FUNCTION_BLOCK fb_Worker
VAR
  _nProcess         : UINT;

  _ItfProcess       : REFERENCE TO ARRAY[1..MAX_PROCESS] OF I_ExternControl_Process;

  _tonProcess       : Tc2_Standard.TON;
  _tProcess         : TIME;

  _nMoverPerMinute  : UINT;

  _wTargetMask      : DWORD;
  _nQueue           : ARRAY[1..MAX_PROCESS] OF UINT;

END_VAR

METHOD AUTO : E_PROGRESS
VAR_INPUT
  Active            : BOOL;
END_VAR
VAR_INST
  _bSparse            : Bool;
  _ncount             : uint;
  _eState,
  _eResult            : E_PROGRESS;

  _ndx                : UINT;

  _eProcessState      : E_STATION_STATE;
  _eProcessCmd        : E_STATION_CTRL;

  _nkx                : UINT;

  _nInputLastTarget   : UINT;

{attribute 'displaymode':='bin'}
  _wBufferSentMask    : dword;
{attribute 'displaymode':='bin'}
  _wProcessInputMask  : dWORD; // placement information for movers in stations from preceeding machine
END_VAR
IF NOT Check() THEN AUTO := E_PROGRESS.PROGRESS_ERROR; RETURN; END_IF

//-----------------------------------------------------------------------------
IF NOT Active 
THEN 
	_eState                                     := E_PROGRESS.PROGRESS_INIT;

  _nCount                                     := 0;
  memset(ADR(_nQueue), 0, SIZEOF(_nQueue));
  memset(ADR(_wProcessInputMask), 0, SIZEOF(_wProcessInputMask));
  memset(ADR(_wBufferSentMask), 0, SIZEOF(_wBufferSentMask));
ELSE
  _eProcessState                              := _ItfProcess[_nProcess].ProcessState;

  FOR _ndx := 1 TO MAX_PROCESS
  DO
    _nQueue[_ndx]                             := _ItfProcess[_ndx].MoverCountInQueue;
  END_FOR
END_IF 
//-----------------------------------------------------------------------------
//-----------------------------------------------------------------------------
//-----------------------------------------------------------------------------
CASE _eState
OF
  E_PROGRESS.PROGRESS_INIT:
    IF Active
    THEN
      _nCount := _ncount + 1;
      _wProcessInputMask                      := 0;
      _wBufferSentMask                        := 0;
      _eState                                 := E_PROGRESS.PROGRESS_BUSY;
    END_IF
END_CASE
//-----------------------------------------------------------------------------
//-----------------------------------------------------------------------------
CASE _eState
OF
  E_PROGRESS.PROGRESS_BUSY:

    CASE _nProcess
    OF
      DISTRIBUTOR_2,
      DISTRIBUTOR_1:
        _eState                               := E_PROGRESS.PROGRESS_PREPARE;

      OUTPUT_R2:
        _eState                               := E_PROGRESS.PROGRESS_PREPARE;

      OUTPUT_R1:
        _eState                               := E_PROGRESS.PROGRESS_PREPARE;

      BUFFER_3:
        IF (_nQueue[BUFFER_3] > QUEUE_COUNT)
        THEN
          _eState                             := E_PROGRESS.PROGRESS_PREPARE;
        END_IF

      OUTPUT_1:
        _eState                               := E_PROGRESS.PROGRESS_PREPARE;

      INPUT:
        _eState                               := E_PROGRESS.PROGRESS_PREPARE;

      BUFFER_1:
        _eState                               := E_PROGRESS.PROGRESS_PREPARE;
        IF NOT _bSparse
        THEN
          FOR _nkx := 1 TO _ItfProcess[INPUT].StationCount
          DO
              _wProcessInputMask              := Tc2_System.SETBIT32(_wProcessInputMask, TO_SINT(_nkx-1));
          END_FOR
        ELSE
          FOR _nkx := 1 TO _ItfProcess[INPUT].StationCount
          DO
            IF (_nkx <> 7)
            THEN
              _wProcessInputMask              := _ItfProcess[BUFFER_1].SetBitDWord(_wProcessInputMask, _nkx-1);
            END_IF
          END_FOR

        END_IF


      BUFFER_4:
        IF (_nQueue[BUFFER_1] < 8)
        THEN
          _eState                             := E_PROGRESS.PROGRESS_PREPARE;
        END_IF
    END_CASE
END_CASE
//-----------------------------------------------------------------------------
//-----------------------------------------------------------------------------
CASE _eState
OF
  E_PROGRESS.PROGRESS_PREPARE:
    CASE _nProcess
    OF
      BUFFER_1:
        _bSparse                              := FALSE;
        IF (_nQueue[INPUT] = 0)
        THEN
          _nInputLastTarget                   := 0;
          _ItfProcess[BUFFER_1].TargetMask    := _wProcessInputMask;
          _eState                             := E_PROGRESS.PROGRESS_WORKING;
        END_IF
    ELSE
      _eState                                 := E_PROGRESS.PROGRESS_WORKING;
    END_CASE

END_CASE
//-----------------------------------------------------------------------------
//-----------------------------------------------------------------------------
CASE _eState
OF
  E_PROGRESS.PROGRESS_WORKING:

  CASE _eProcessState
  OF
    E_STATION_STATE.STATION_INIT:
      CASE _nProcess
      OF
        BUFFER_3:
          IF (_nQueue[OUTPUT_R1] = QUEUE_COUNT)
          THEN
            _eState                           := E_PROGRESS.PROGRESS_INIT;
          ELSE
            _eProcessCmd                      := E_STATION_CTRL.STATION_DISABLE;
          END_IF
      ELSE
        _eProcessCmd                          := E_STATION_CTRL.STATION_DISABLE;
      END_CASE

    E_STATION_STATE.STATION_DISABLE:
      _eProcessCmd                            := E_STATION_CTRL.STATION_ENABLE;

    E_STATION_STATE.STATION_MOVER_ENTER:
      CASE _ItfProcess[_nProcess].ProcessType
      OF
        E_PROCESS_TYPE.DISTRIBUTOR:
          IF (GVL_XTS.StationState[_ItfProcess[_nProcess].StationFirst].rMoverModPos > GVL_XTS.StationParameter[_ItfProcess[_nProcess].StationFirst].rPosWait-5.0)
          THEN
            _eState                           := E_PROGRESS.PROGRESS_OCCUPIED;
            _eProcessCmd                      := E_STATION_CTRL.STATION_MOVER_SEND;
          END_IF
      ELSE
          _eProcessCmd                        := E_STATION_CTRL.STATION_MOVER_ENTER;
      END_CASE

    E_STATION_STATE.STATION_PROCESS_START:
      _tonProcess(IN := FALSE, PT := _tProcess);
      CASE _nProcess
      OF
        INPUT:
          IF (_nQueue[INPUT] = QUEUE_COUNT)
          THEN
            _eProcessCmd                      := E_STATION_CTRL.STATION_PROCESS_START;
          END_IF

        OUTPUT_R1,
        OUTPUT_R2:
          IF (_ItfProcess[OUTPUT_R1].ProcessState = _ItfProcess[OUTPUT_R2].ProcessState)
          THEN
            _eProcessCmd                      := E_STATION_CTRL.STATION_PROCESS_START;
          END_IF
      ELSE
        _eProcessCmd                          := E_STATION_CTRL.STATION_PROCESS_START;
      END_CASE


    E_STATION_STATE.STATION_PROCESS_DONE:
      _tonProcess(IN := TRUE, PT := _tProcess);

      IF _tonProcess.Q
      THEN
        _eProcessCmd                          := E_STATION_CTRL.STATION_PROCESS_DONE;
      END_IF

    E_STATION_STATE.STATION_MOVER_OUT:
      CASE _nProcess
      OF
        BUFFER_1:
          _eState                             := E_PROGRESS.PROGRESS_CHECK;

        Buffer_4:
          _eProcessCmd                        := E_STATION_CTRL.STATION_MOVER_OUT;
          IF (_nQueue[BUFFER_1] = QUEUE_COUNT-1)
          THEN
            _eState                           := E_PROGRESS.PROGRESS_INIT;
          END_IF

        BUFFER_3: 
          _eProcessCmd                        := E_STATION_CTRL.STATION_MOVER_OUT;


        OUTPUT_R1,
        OUTPUT_R2:
          IF (_ItfProcess[OUTPUT_R1].ProcessState = E_STATION_STATE.STATION_MOVER_OUT) AND
             (_ItfProcess[OUTPUT_R2].ProcessState = E_STATION_STATE.STATION_MOVER_OUT)
          THEN
            _eState                           := E_PROGRESS.PROGRESS_INIT;
            _eProcessCmd                      := E_STATION_CTRL.STATION_MOVER_OUT;
          END_IF

      ELSE
          _eState                             := E_PROGRESS.PROGRESS_INIT;
          _eProcessCmd                        := E_STATION_CTRL.STATION_MOVER_OUT;
      END_CASE
  END_CASE

END_CASE
//-----------------------------------------------------------------------------
//-----------------------------------------------------------------------------
CASE _eState
OF
  E_PROGRESS.PROGRESS_OCCUPIED:
      CASE _nProcess
      OF
        BUFFER_1:
          CASE _eProcessState
          OF
            E_STATION_STATE.STATION_MOVER_OUT:
            _wBufferSentMask                  := _ItfProcess[_nProcess].SetBitDWord(_wBufferSentMask, _nInputLastTarget);
            _nInputLastTarget                 := _nInputLastTarget + 1;
            _eState                           := E_PROGRESS.PROGRESS_WORKING;
          END_CASE
      ELSE
        _eState                               := E_PROGRESS.PROGRESS_WORKING;
      END_CASE
END_CASE
//-----------------------------------------------------------------------------
//-----------------------------------------------------------------------------
CASE _eState
OF
  E_PROGRESS.PROGRESS_CHECK:
    CASE _nProcess
    OF
      BUFFER_1:
        _eProcessCmd                          := E_STATION_CTRL.STATION_MOVER_OUT;
        IF (_wBufferSentMask = _wProcessInputMask)
        THEN
          _eState                             := E_PROGRESS.PROGRESS_INIT;
        ELSE
          _eState                             := E_PROGRESS.PROGRESS_WORKING;
        END_IF
    ELSE
      _eState                                 := E_PROGRESS.PROGRESS_INIT;
    END_CASE
END_CASE
//-----------------------------------------------------------------------------
//-----------------------------------------------------------------------------
_ItfProcess[_nProcess].ProcessCmd             := _eProcessCmd; 
AUTO                                          := _eState;
//-----------------------------------------------------------------------------
//-----------------------------------------------------------------------------
END_METHOD

METHOD AUTO_1 : E_PROGRESS
VAR_INPUT
  Active            : BOOL;
END_VAR
VAR_INST
  _bSparse            : Bool;
  _ncount             : uint;
  _eState,
  _eResult            : E_PROGRESS;

  _ndx                : UINT;

  _eProcessState      : E_STATION_STATE;
  _eProcessCmd        : E_STATION_CTRL;

  _nkx                : UINT;

  _nInputLastTarget   : UINT;

{attribute 'displaymode':='bin'}
  _wBufferSentMask    : dword;
{attribute 'displaymode':='bin'}
  _wProcessInputMask  : DWORD; // placement information for movers in stations from preceeding machine

  _eProcessType       : E_PROCESS_TYPE;
END_VAR
IF NOT Check() THEN AUTO_1 := E_PROGRESS.PROGRESS_ERROR; RETURN; END_IF

//-----------------------------------------------------------------------------
IF NOT Active 
THEN 
	_eState                                     := E_PROGRESS.PROGRESS_INIT;

  _nCount                                     := 0;
  memset(ADR(_nQueue), 0, SIZEOF(_nQueue));
  memset(ADR(_wProcessInputMask), 0, SIZEOF(_wProcessInputMask));
  memset(ADR(_wBufferSentMask), 0, SIZEOF(_wBufferSentMask));
ELSE
  _eProcessState                              := _ItfProcess[_nProcess].ProcessState;
  _eProcessType                               := _ItfProcess[_nProcess].ProcessType;

  FOR _ndx := 1 TO MAX_PROCESS
  DO
    _nQueue[_ndx]                             := _ItfProcess[_ndx].MoverCountInQueue;
  END_FOR
END_IF 
//-----------------------------------------------------------------------------
//-----------------------------------------------------------------------------
//-----------------------------------------------------------------------------
CASE _eState
OF
  E_PROGRESS.PROGRESS_INIT:
    IF Active
    THEN
      _nCount := _ncount + 1;
      _wProcessInputMask                      := 0;
      _wBufferSentMask                        := 0;
      _eState                                 := E_PROGRESS.PROGRESS_BUSY;
    END_IF
END_CASE
//-----------------------------------------------------------------------------
//-----------------------------------------------------------------------------
CASE _eState
OF
  E_PROGRESS.PROGRESS_BUSY:

    CASE _nProcess
    OF
      DISTRIBUTOR_2,
      DISTRIBUTOR_1:
        _eState                               := E_PROGRESS.PROGRESS_PREPARE;

      OUTPUT_R2:
        _eState                               := E_PROGRESS.PROGRESS_PREPARE;

      OUTPUT_R1:
        _eState                               := E_PROGRESS.PROGRESS_PREPARE;

      BUFFER_3:
        IF (_nQueue[_nProcess] > 11)
        THEN
          _eState                             := E_PROGRESS.PROGRESS_PREPARE;
        END_IF

      OUTPUT_1:
        _eState                               := E_PROGRESS.PROGRESS_PREPARE;

      INPUT:
        _eState                               := E_PROGRESS.PROGRESS_PREPARE;

      BUFFER_1:
        _eState                               := E_PROGRESS.PROGRESS_PREPARE;
        IF NOT _bSparse
        THEN
          FOR _nkx := 1 TO _ItfProcess[INPUT].StationCount
          DO
              _wProcessInputMask              := _ItfProcess[BUFFER_1].SetBitDWord(_wProcessInputMask, _nkx-1);
          END_FOR
        ELSE
          FOR _nkx := 1 TO _ItfProcess[INPUT].StationCount
          DO
            IF (_nkx <> 7)
            THEN
              _wProcessInputMask              := _ItfProcess[BUFFER_1].SetBitDWord(_wProcessInputMask, _nkx-1);
            END_IF
          END_FOR

        END_IF


      BUFFER_4:
        IF (_nQueue[BUFFER_1] < 8)
        THEN
          _eState                             := E_PROGRESS.PROGRESS_PREPARE;
        END_IF
    END_CASE
END_CASE
//-----------------------------------------------------------------------------
//-----------------------------------------------------------------------------
CASE _eState
OF
  E_PROGRESS.PROGRESS_PREPARE:
    CASE _nProcess
    OF
      BUFFER_1:
        _bSparse                              := FALSE;
        IF (_nQueue[INPUT] = 0)
        THEN
          _nInputLastTarget                   := 0;
          _ItfProcess[BUFFER_1].TargetMask    := _wProcessInputMask;
          _eState                             := E_PROGRESS.PROGRESS_WORKING;
        END_IF
    ELSE
      _eState                                 := E_PROGRESS.PROGRESS_WORKING;
    END_CASE

END_CASE
//-----------------------------------------------------------------------------
//-----------------------------------------------------------------------------
CASE _eState
OF
  E_PROGRESS.PROGRESS_WORKING:

  CASE _eProcessState
  OF
    E_STATION_STATE.STATION_INIT:
      _eProcessCmd                            := E_STATION_CTRL.STATION_DISABLE;

    E_STATION_STATE.STATION_DISABLE:
      _eProcessCmd                            := E_STATION_CTRL.STATION_ENABLE;

    E_STATION_STATE.STATION_MOVER_ENTER:
      CASE _eProcessType
      OF
        E_PROCESS_TYPE.DISTRIBUTOR:
          IF (GVL_XTS.StationState[_ItfProcess[_nProcess].StationFirst].rMoverModPos > GVL_XTS.StationParameter[_ItfProcess[_nProcess].StationFirst].rPosWait - 250.0)
          THEN
            _eState                           := E_PROGRESS.PROGRESS_OCCUPIED;
            _eProcessCmd                      := E_STATION_CTRL.STATION_MOVER_SEND;
          END_IF
      ELSE
          _eProcessCmd                        := E_STATION_CTRL.STATION_MOVER_ENTER;
      END_CASE

    E_STATION_STATE.STATION_PROCESS_START:
      _tonProcess(IN := FALSE, PT := _tProcess);
      _eProcessCmd                            := E_STATION_CTRL.STATION_PROCESS_START;


    E_STATION_STATE.STATION_PROCESS_DONE:
      _tonProcess(IN := TRUE, PT := _tProcess);

      IF _tonProcess.Q
      THEN
        _eProcessCmd                          := E_STATION_CTRL.STATION_PROCESS_DONE;
      END_IF

    E_STATION_STATE.STATION_MOVER_OUT:
      CASE _nProcess
      OF
        BUFFER_1:
          _eState                             := E_PROGRESS.PROGRESS_CHECK;

        Buffer_4:
          _eProcessCmd                        := E_STATION_CTRL.STATION_MOVER_OUT;
          IF (_nQueue[BUFFER_1] = QUEUE_COUNT-1)
          THEN
            _eState                           := E_PROGRESS.PROGRESS_INIT;
          END_IF

        BUFFER_3: 
          _eProcessCmd                        := E_STATION_CTRL.STATION_MOVER_OUT;
          IF (_nQueue[OUTPUT_R1] = QUEUE_COUNT)
          THEN
            _eState                           := E_PROGRESS.PROGRESS_INIT;
          END_IF


      ELSE
          _eState                             := E_PROGRESS.PROGRESS_INIT;
          _eProcessCmd                        := E_STATION_CTRL.STATION_MOVER_OUT;
      END_CASE
  END_CASE

END_CASE
//-----------------------------------------------------------------------------
//-----------------------------------------------------------------------------
CASE _eState
OF
  E_PROGRESS.PROGRESS_OCCUPIED:
      CASE _nProcess
      OF
        BUFFER_1:
          CASE _eProcessState
          OF
            E_STATION_STATE.STATION_MOVER_OUT:
            _wBufferSentMask                  := _ItfProcess[_nProcess].SetBitDWord(_wBufferSentMask, _nInputLastTarget);
            _nInputLastTarget                 := _nInputLastTarget + 1;
            _eState                           := E_PROGRESS.PROGRESS_WORKING;
          END_CASE
      ELSE
        _eState                               := E_PROGRESS.PROGRESS_WORKING;
      END_CASE
END_CASE
//-----------------------------------------------------------------------------
//-----------------------------------------------------------------------------
CASE _eState
OF
  E_PROGRESS.PROGRESS_CHECK:
    CASE _nProcess
    OF
      BUFFER_1:
        _eProcessCmd                          := E_STATION_CTRL.STATION_MOVER_OUT;
        IF (_wBufferSentMask = _wProcessInputMask)
        THEN
          _ItfProcess[BUFFER_1].TargetMask    := 0;
          _eState                             := E_PROGRESS.PROGRESS_INIT;
        ELSE
          _eState                             := E_PROGRESS.PROGRESS_WORKING;
        END_IF
    ELSE
      _eState                                 := E_PROGRESS.PROGRESS_INIT;
    END_CASE
END_CASE
//-----------------------------------------------------------------------------
//-----------------------------------------------------------------------------
_ItfProcess[_nProcess].ProcessCmd             := _eProcessCmd; 
AUTO_1                                          := _eState;
//-----------------------------------------------------------------------------
//-----------------------------------------------------------------------------
END_METHOD

METHOD Check : BOOL
VAR_INST
  _sCheck   : STRING;
  _nIdx     : UINT;
END_VAR

FOR _nIdx := 1 TO MAX_PROCESS
DO
  IF NOT (_ItfProcess[_nIdx] <> 0)
  THEN
    _sCheck   := concat('Invalid Interface Pointer at Index: ', TO_STRING(_nIdx));
    RETURN;
  END_IF
END_FOR

IF NOT (_nProcess > 0)
THEN
  _sCheck         := concat('NULL Invalid Index: ', TO_STRING(_nProcess));
  RETURN;
END_IF

IF (_nProcess > MAX_PROCESS)
THEN
  _sCheck         := concat('MAX Invalid Index: ', TO_STRING(_nProcess));
  RETURN;
END_IF

_nMoverPerMinute  := _ItfProcess[_nProcess].ProcessPerMinute;
_wTargetMask      := _ItfProcess[_nProcess].TargetMask;

Check             := TRUE;
END_METHOD

PROPERTY ItfProcesses : reference to ARRAY[1..MAX_PROCESS] OF I_ExternControl_Process
SET
_ItfProcess REF= ItfProcesses;
END_SET
END_PROPERTY

PROPERTY ProcessIndex : uint
GET
ProcessIndex  := _nProcess;
END_GET
SET
_nProcess   := ProcessIndex;
END_SET
END_PROPERTY

PROPERTY ProcessTime : time
GET
ProcessTime := _tProcess;
END_GET
SET
_tProcess := ProcessTime;
END_SET
END_PROPERTY

METHOD RESET : E_PROGRESS
VAR_INPUT
  Execute         : BOOL;
END_VAR
VAR
  _eState,
  _eResult          : E_PROGRESS;
END_VAR

//-----------------------------------------------------------------------------
IF NOT Execute 
THEN 
	_eState                                     := E_PROGRESS.PROGRESS_INIT; 
END_IF 
//-----------------------------------------------------------------------------
//-----------------------------------------------------------------------------
//-----------------------------------------------------------------------------
CASE _eState
OF
  E_PROGRESS.PROGRESS_INIT:
    IF Execute
    THEN
      IF NOT (_ItfProcess[_nProcess] <> 0)
      THEN
        _eState                               := E_PROGRESS.PROGRESS_ERROR;
      ELSE
        _eState                               := E_PROGRESS.PROGRESS_BUSY;
      END_IF
    END_IF
END_CASE
//-----------------------------------------------------------------------------
//-----------------------------------------------------------------------------
CASE _eState
OF
  E_PROGRESS.PROGRESS_BUSY:
    _eState                                   := E_PROGRESS.PROGRESS_PREPARE;
END_CASE
//-----------------------------------------------------------------------------
//-----------------------------------------------------------------------------
CASE _eState
OF
  E_PROGRESS.PROGRESS_PREPARE:
    IF (_ItfProcess[_nProcess].Init())
    THEN
      _eState                                 := E_PROGRESS.PROGRESS_DONE;
    END_IF
END_CASE
//-----------------------------------------------------------------------------
//-----------------------------------------------------------------------------
END_METHOD

END_FUNCTION_BLOCK

(* stored: Version 1.1.0.1, ProductVersion 3.1.4024.12
   POU fb_Worker: Id {9c4c4670-648c-4781-a655-54f8931867d3}, SpecialFunc None
   Folder private: Id {4ff00cee-edd5-446f-b1e2-d6539cc999ce}
   Folder properties: Id {63012438-1888-49c9-a937-dba53dd37d80}
   Folder public: Id {101027a7-9274-4a18-8032-86265a759e66}
   Method AUTO: Id {cdf26a9c-fe5d-49bd-917d-9a453e096f46}
   Method AUTO_1: Id {14635e9b-9edf-4af9-ae26-6b129c13e362}
   Method Check: Id {9c3da242-113a-4e35-8d07-6d7d0c14a6f9}
   Property ItfProcesses: Id {d644fffd-7506-4ce5-9112-0308a862c0fb}
   Set Set: Id {d4304595-6288-48a2-b012-572851462ba3}
   Property ProcessIndex: Id {0595c6ae-05b0-41f0-a1d5-8a89918040f2}
   Get Get: Id {03e2c372-05db-407c-92be-8e0de95655f1}
   Set Set: Id {7ef33abc-632d-49ce-8b75-3a0475a9c174}
   Property ProcessTime: Id {4eae8ecb-b4f4-449a-865c-8601ed5dbb30}
   Get Get: Id {ee6d1d7f-d429-44d6-b122-b23a11df00ff}
   Set Set: Id {2791910b-23e8-45e7-b0e1-d7c5c3f7114e}
   Method RESET: Id {1fb32989-6ae4-40ab-b359-0e8b0ae000bc} *)
